(* PLC project PLC, Beckhoff Automation GmbH TwinCAT PLC Control 3.5.13.21 *)
(* stored: creationDateTime 2024-02-17T22:43:28.8590095, modificationDateTime 2024-02-17T22:43:28.8590095 *)

FUNCTION_BLOCK Cyl
VAR_INPUT
	index: LINT;
	name: STRING(G.nameStringLength);
	opeFw: BOOL;
	opeRv: BOOL;
END_VAR
VAR_OUTPUT
	posFw: BOOL;
	posRv: BOOL;
	ready: BOOL;
	busy: BOOL;
	done: BOOL;
	error: BOOL;
END_VAR
VAR_IN_OUT
	resources: ARRAY[0..G.numAxis] OF CylResource;
END_VAR
VAR
	input: CylInput;
	output: CylOutput;
	config: CylConfig;
	status: CylStatus;
	rsErrorON: BOOL;
	rsErrorOFF: BOOL;
	cylErrorFw: BOOL;
	cylErrorRv: BOOL;
	TON_0: TON;
	TON_1: TON;
	TON_2: TON;
	TON_3: TON;
	TON_4: TON;
	TON_5: TON;
END_VAR

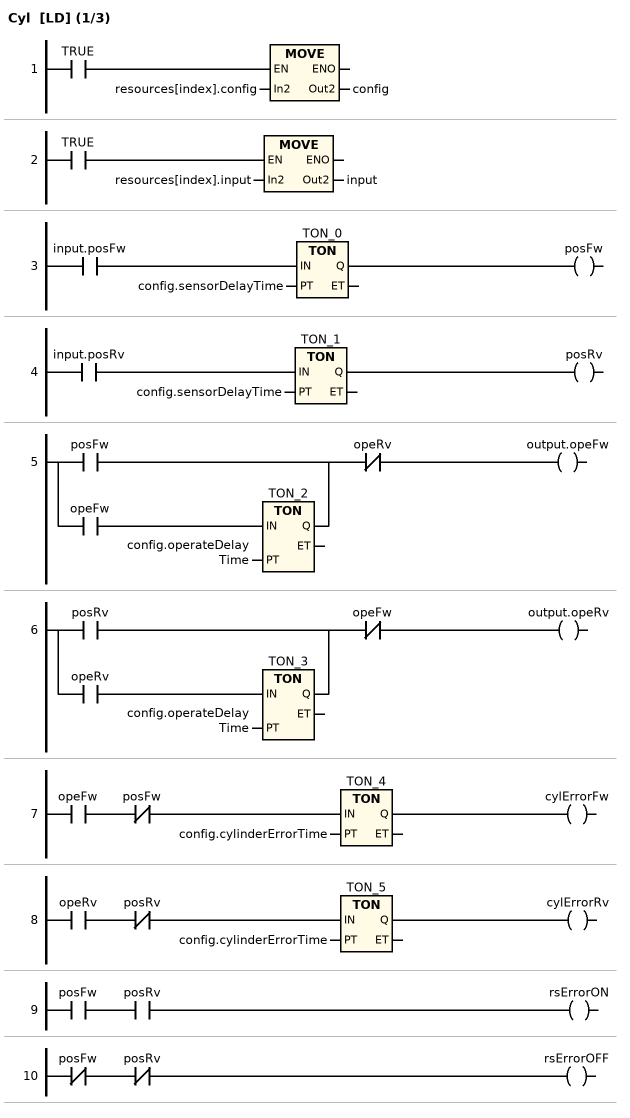
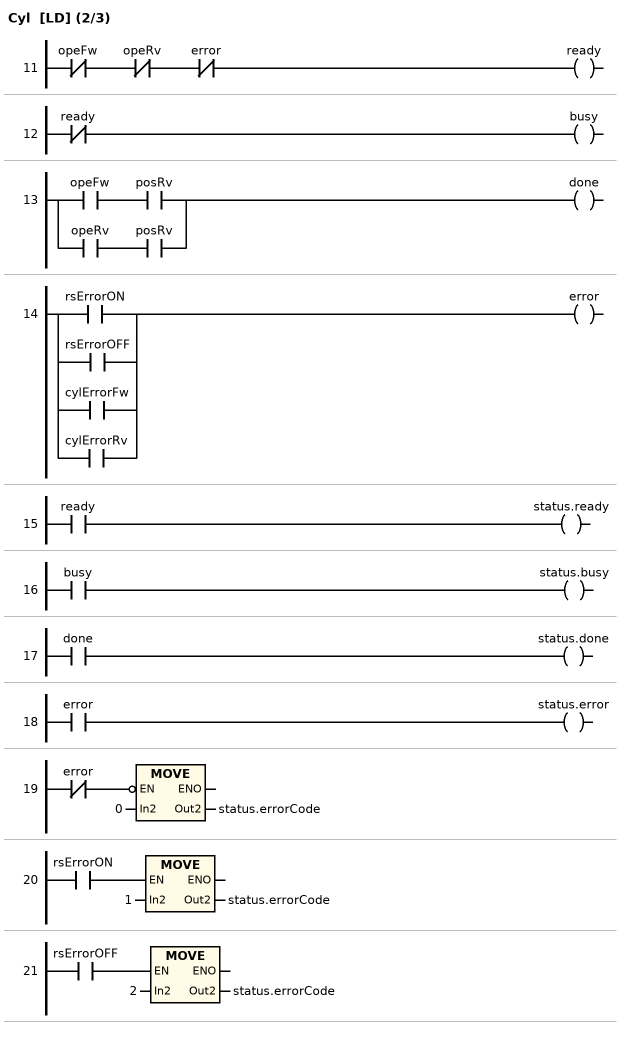
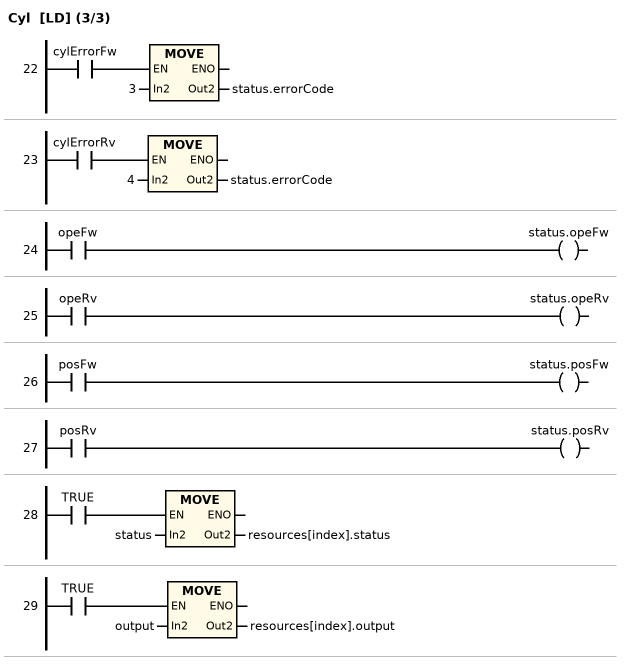
(* LD diagram, written out as Structured Text *)

IF TRUE THEN config := resources[index].config; END_IF;

IF TRUE THEN input := resources[index].input; END_IF;

TON_0(IN := input.posFw, PT := config.sensorDelayTime);
posFw := TON_0.Q;

TON_1(IN := input.posRv, PT := config.sensorDelayTime);
posRv := TON_1.Q;

TON_2(IN := opeFw, PT := config.operateDelayTime);
output.opeFw := (TON_2.Q OR posFw) AND NOT opeRv;

TON_3(IN := opeRv, PT := config.operateDelayTime);
output.opeRv := (TON_3.Q OR posRv) AND NOT opeFw;

TON_4(IN := opeFw AND NOT posFw, PT := config.cylinderErrorTime);
cylErrorFw := TON_4.Q;

TON_5(IN := opeRv AND NOT posRv, PT := config.cylinderErrorTime);
cylErrorRv := TON_5.Q;

rsErrorON := posFw AND posRv;

rsErrorOFF := NOT posFw AND NOT posRv;

ready := NOT opeFw AND NOT opeRv AND NOT error;

busy := NOT ready;

done := opeFw AND posRv OR opeRv AND posRv;

error := rsErrorON OR rsErrorOFF OR cylErrorFw OR cylErrorRv;

status.ready := ready;

status.busy := busy;

status.done := done;

status.error := error;

IF NOT (NOT error) THEN status.errorCode := 0; END_IF;

IF rsErrorON THEN status.errorCode := 1; END_IF;

IF rsErrorOFF THEN status.errorCode := 2; END_IF;

IF cylErrorFw THEN status.errorCode := 3; END_IF;

IF cylErrorRv THEN status.errorCode := 4; END_IF;

status.opeFw := opeFw;

status.opeRv := opeRv;

status.posFw := posFw;

status.posRv := posRv;

IF TRUE THEN resources[index].status := status; END_IF;

IF TRUE THEN resources[index].output := output; END_IF;
(* --- network --- *)
END_FUNCTION_BLOCK
